FUNCTION IsEqualAnyType : E_GeneralResult
VAR_INPUT
	A					: __SYSTEM.AnyType; // A and B have to be same type
	B					: __SYSTEM.AnyType; // A and B have to be same type
END_VAR
VAR
	isEqual				: BOOL;
END_VAR


IF A.TypeClass <> B.TypeClass THEN

	RETURN;
END_IF

isEqual := MEMCMP(A.pValue, B.pValue, A.diSize) = 0;

IF isEqual THEN

	IsEqualAnyType := E_GeneralResult._TRUE;
ELSE

	IsEqualAnyType := E_GeneralResult._FALSE;
END_IF

END_FUNCTION

(* stored: Version 1.1.0.1, ProductVersion 3.1.4024.11
   POU IsEqualAnyType: Id {0c403136-e827-45c6-a5a8-7d1320cc8888}, SpecialFunc None *)
